Omron CX-Programmer project NewProject (CX-Programmer 9.70)

# PLC NOVO_PAP: CP1L-E EM

## Program NewProgram1 (cyclic task 0)
; POS0
Local symbols
ABRIR_LIQUIDO1 205.00 BOOL
ABRIR_LIQUIDO2 205.01 BOOL  ; ~
ABRIR_LIQUIDO3 205.02 BOOL
BIT_EXTRA1_IN 1.02 BOOL
BIT_EXTRA1_OUT 100.03 BOOL
BIT_EXTRA2_IN 1.03 BOOL
BIT_EXTRA2_OUT 100.06 BOOL
BUSY 0.06 BOOL
CONDICAO 207.01 BOOL
ENTR_1 0.07 BOOL
ENTR_2 0.08 BOOL
ENTR_3 0.09 BOOL
ENTR_4 0.10 BOOL
ENTR_5 0.11 BOOL
ENTR_6 1.00 BOOL
ENTR_7 1.01 BOOL
ENVIAR100 101.03 BOOL
ENVIAR33 101.00 BOOL
ENVIAR50 101.01 BOOL
ENVIAR66 101.02 BOOL
ENVIAR_ROBO 100.05 BOOL
ET BOOL
ET0 200.00 BOOL
ET10 200.01 BOOL  ; SVON
ET100 203.00 BOOL
ET110 203.01 BOOL
ET120 203.02 BOOL
ET130 203.03 BOOL
ET140 203.04 BOOL
ET150 203.05 BOOL
ET160 203.06 BOOL
ET170 203.07 BOOL
ET20 200.02 BOOL  ; SETUP
ET200 203.00 BOOL
ET210 203.01 BOOL
ET220 203.02 BOOL
ET230 203.03 BOOL
ET240 203.04 BOOL
ET250 203.05 BOOL
ET260 203.06 BOOL
ET30 200.03 BOOL
ET40 200.04 BOOL
ET50 200.05 BOOL
ET60 200.06 BOOL
ET70 200.07 BOOL
ET80 201.00 BOOL
ET_POS0 202.00 BOOL
ET_POS1 202.01 BOOL
ET_POS2 202.02 BOOL
ET_POS_RETORNO 202.05 BOOL
EXTRA_BIT1_IN BOOL
FAKE_IMPULSO 201.01 BOOL
IMPULSO 100.02 BOOL
IN0 100.01 BOOL
IN0W 202.03 BOOL
IN1 100.00 BOOL
IN1W 202.04 BOOL
IS_WORKING 207.02 BOOL
JA_TEM_VALOR1 203.07 BOOL
JA_TEM_VALOR2 204.04 BOOL
JA_TEM_VALOR3 204.05 BOOL
LIQUIDO1 D20 INT
LIQUIDO2 D21 INT
LIQUIDO3 D22 INT
MULT_1 D10 UINT
MULT_2 D11 UINT
MULT_3 D12 UINT
MULT_4 D13 UINT
MULT_5 D14 UINT
MULT_6 D15 UINT
MULT_7 D16 UINT
M_START 207.00 BOOL
M_STARt BOOL
NUM100 204.03 BOOL
NUM33 204.00 BOOL
NUM50 204.01 BOOL
NUM66 204.02 BOOL
OUT0 0.03 BOOL
OUT1 0.02 BOOL
POS0 201.02 BOOL
POS1 201.03 BOOL
POS1_TIMER 201.06 BOOL
POS2 201.04 BOOL
POS2_TIMER 201.07 BOOL
POS3 BOOL
POS_RASP 1.04 BOOL
POS_RASP2 1.05 BOOL
POS_RETORNO 201.05 BOOL
SETON 0.04 BOOL
SETUP 100.07 BOOL
START 0.01 BOOL
STOP 0.00 BOOL
SVON 100.04 BOOL
Start_Virtual 5.01 BOOL

### Section MAIN

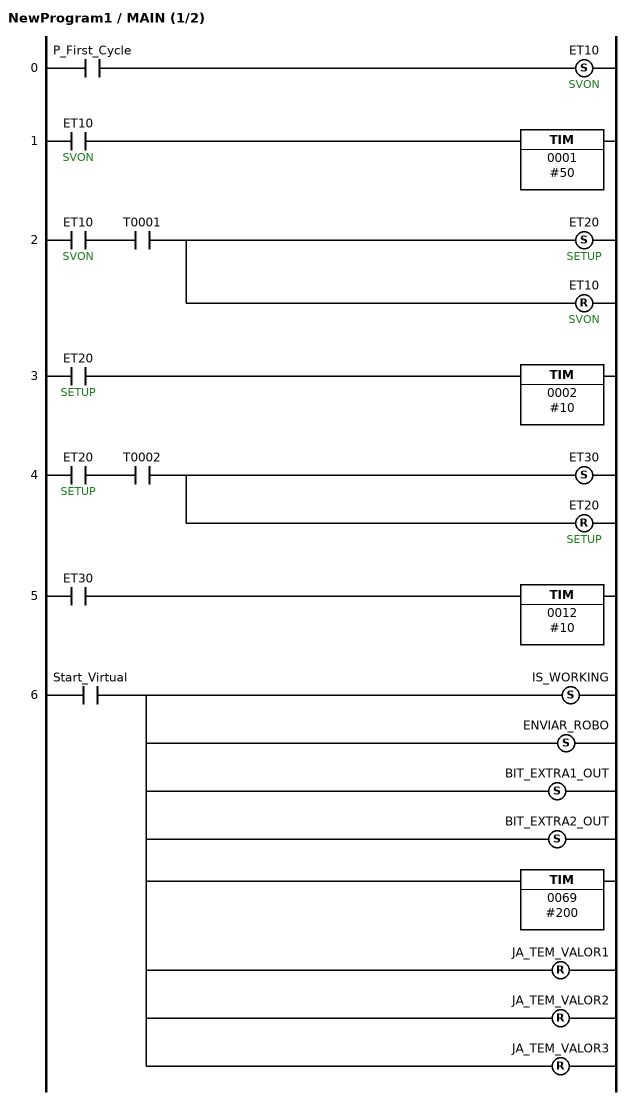
; rung 0
LD P_First_Cycle
SET ET10  ; SVON
; rung 1
LD ET10  ; SVON
TIM 0001 #50
; rung 2
LD ET10  ; SVON
AND T0001
SET ET20  ; SETUP
RSET ET10  ; SVON
; rung 3
LD ET20  ; SETUP
TIM 0002 #10
; rung 4
LD ET20  ; SETUP
AND T0002
SET ET30
RSET ET20  ; SETUP
; rung 5
LD ET30
TIM 0012 #10
; rung 6
LD Start_Virtual
SET IS_WORKING
SET ENVIAR_ROBO
SET BIT_EXTRA1_OUT
SET BIT_EXTRA2_OUT
TIM 0069 #200
RSET JA_TEM_VALOR1
RSET JA_TEM_VALOR2
RSET JA_TEM_VALOR3

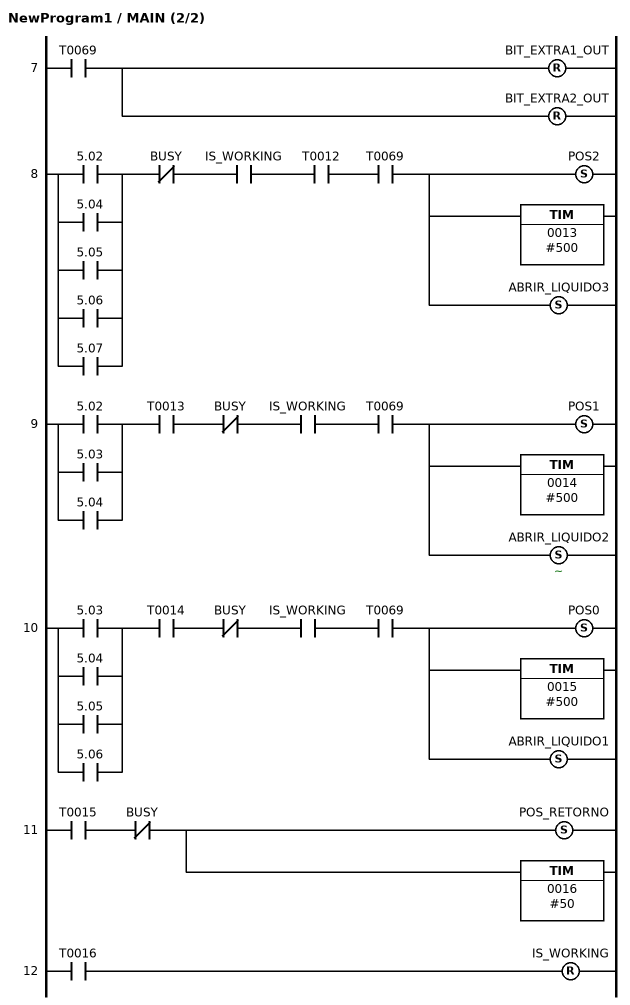
; rung 7
LD T0069
RSET BIT_EXTRA1_OUT
RSET BIT_EXTRA2_OUT
; rung 8
LD 5.02
OR 5.04
OR 5.05
OR 5.06
OR 5.07
ANDNOT BUSY
AND IS_WORKING
AND T0012
AND T0069
SET POS2
TIM 0013 #500
SET ABRIR_LIQUIDO3
; rung 9
LD 5.02
OR 5.03
OR 5.04
AND T0013
ANDNOT BUSY
AND IS_WORKING
AND T0069
SET POS1
TIM 0014 #500
SET ABRIR_LIQUIDO2  ; ~
; rung 10
LD 5.03
OR 5.04
OR 5.05
OR 5.06
AND T0014
ANDNOT BUSY
AND IS_WORKING
AND T0069
SET POS0
TIM 0015 #500
SET ABRIR_LIQUIDO1
; rung 11
LD T0015
ANDNOT BUSY
SET POS_RETORNO
TIM 0016 #50
; rung 12
LD T0016
RSET IS_WORKING

### Section SAIDAS

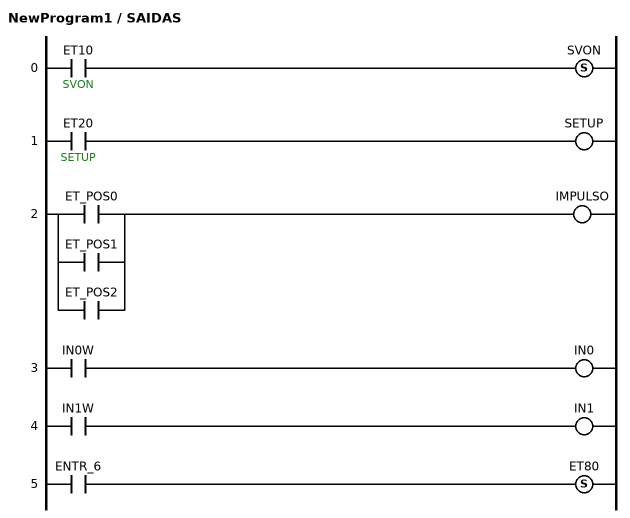
; rung 0
LD ET10  ; SVON
SET SVON
; rung 1
LD ET20  ; SETUP
OUT SETUP
; rung 2
LD ET_POS0
OR ET_POS1
OR ET_POS2
OUT IMPULSO
; rung 3
LD IN0W
OUT IN0
; rung 4
LD IN1W
OUT IN1
; rung 5
LD ENTR_6
SET ET80

### Section DE_RASP

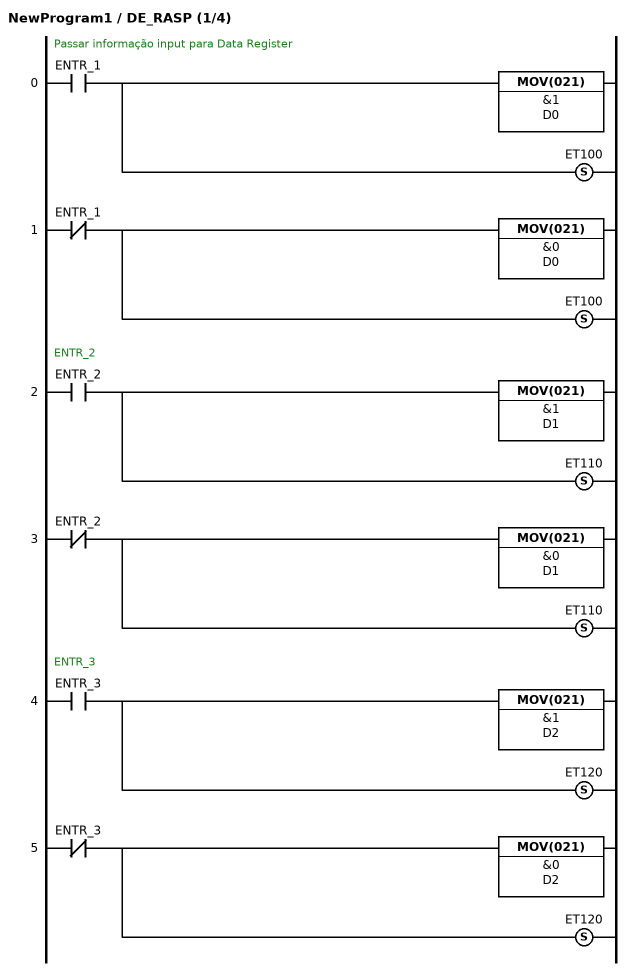
; rung 0: Passar informação input para Data Register
LD ENTR_1
MOV(021) &1 D0
SET ET100
; rung 1
LDNOT ENTR_1
MOV(021) &0 D0
SET ET100
; rung 2: ENTR_2
LD ENTR_2
MOV(021) &1 D1
SET ET110
; rung 3
LDNOT ENTR_2
MOV(021) &0 D1
SET ET110
; rung 4: ENTR_3
LD ENTR_3
MOV(021) &1 D2
SET ET120
; rung 5
LDNOT ENTR_3
MOV(021) &0 D2
SET ET120

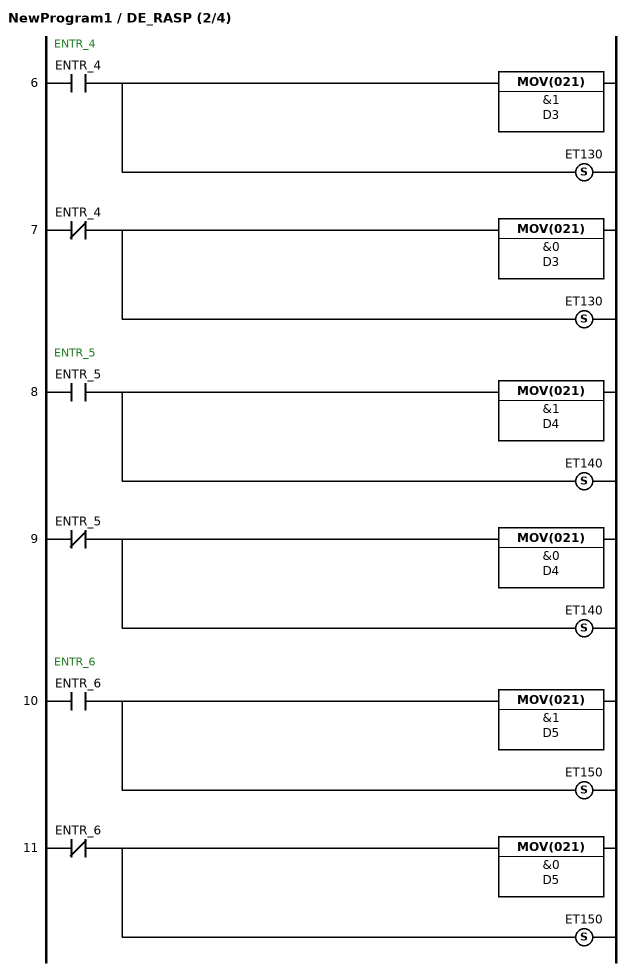
; rung 6: ENTR_4
LD ENTR_4
MOV(021) &1 D3
SET ET130
; rung 7
LDNOT ENTR_4
MOV(021) &0 D3
SET ET130
; rung 8: ENTR_5
LD ENTR_5
MOV(021) &1 D4
SET ET140
; rung 9
LDNOT ENTR_5
MOV(021) &0 D4
SET ET140
; rung 10: ENTR_6
LD ENTR_6
MOV(021) &1 D5
SET ET150
; rung 11
LDNOT ENTR_6
MOV(021) &0 D5
SET ET150

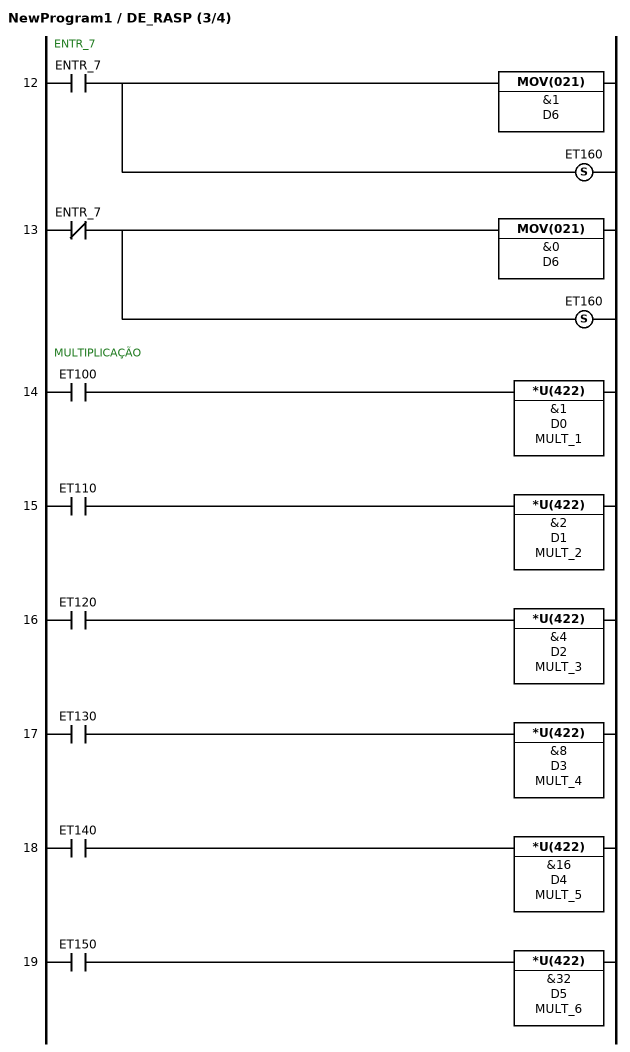
; rung 12: ENTR_7
LD ENTR_7
MOV(021) &1 D6
SET ET160
; rung 13
LDNOT ENTR_7
MOV(021) &0 D6
SET ET160
; rung 14: MULTIPLICAÇÃO
LD ET100
*U(422) &1 D0 MULT_1
; rung 15
LD ET110
*U(422) &2 D1 MULT_2
; rung 16
LD ET120
*U(422) &4 D2 MULT_3
; rung 17
LD ET130
*U(422) &8 D3 MULT_4
; rung 18
LD ET140
*U(422) &16 D4 MULT_5
; rung 19
LD ET150
*U(422) &32 D5 MULT_6

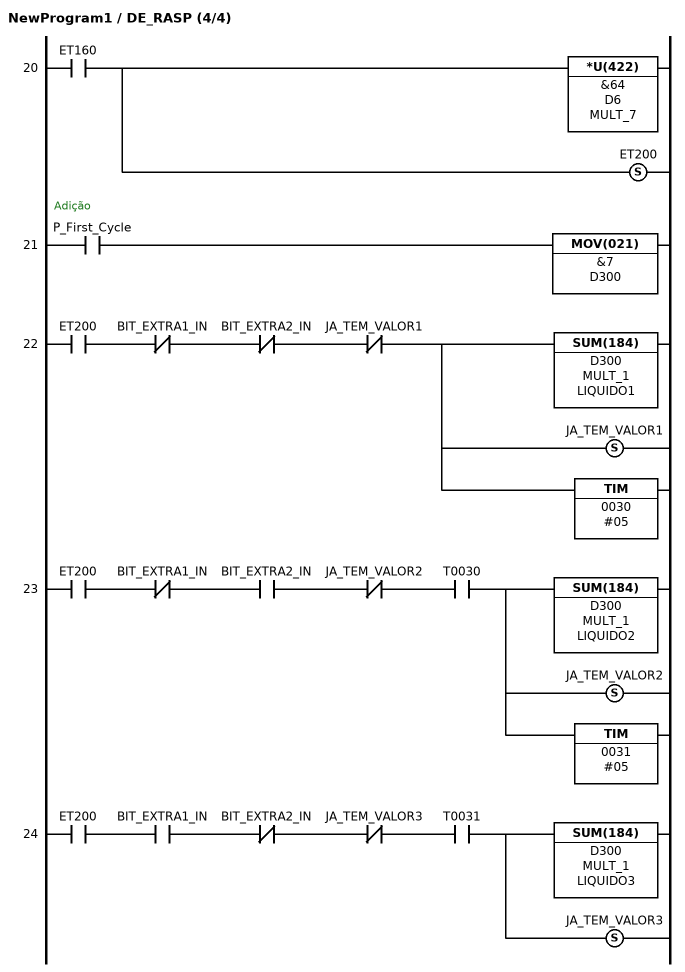
; rung 20
LD ET160
*U(422) &64 D6 MULT_7
SET ET200
; rung 21: Adição
LD P_First_Cycle
MOV(021) &7 D300
; rung 22
LD ET200
ANDNOT BIT_EXTRA1_IN
ANDNOT BIT_EXTRA2_IN
ANDNOT JA_TEM_VALOR1
SUM(184) D300 MULT_1 LIQUIDO1
SET JA_TEM_VALOR1
TIM 0030 #05
; rung 23
LD ET200
ANDNOT BIT_EXTRA1_IN
AND BIT_EXTRA2_IN
ANDNOT JA_TEM_VALOR2
AND T0030
SUM(184) D300 MULT_1 LIQUIDO2
SET JA_TEM_VALOR2
TIM 0031 #05
; rung 24
LD ET200
AND BIT_EXTRA1_IN
ANDNOT BIT_EXTRA2_IN
ANDNOT JA_TEM_VALOR3
AND T0031
SUM(184) D300 MULT_1 LIQUIDO3
SET JA_TEM_VALOR3

### Section POSIÇÕES

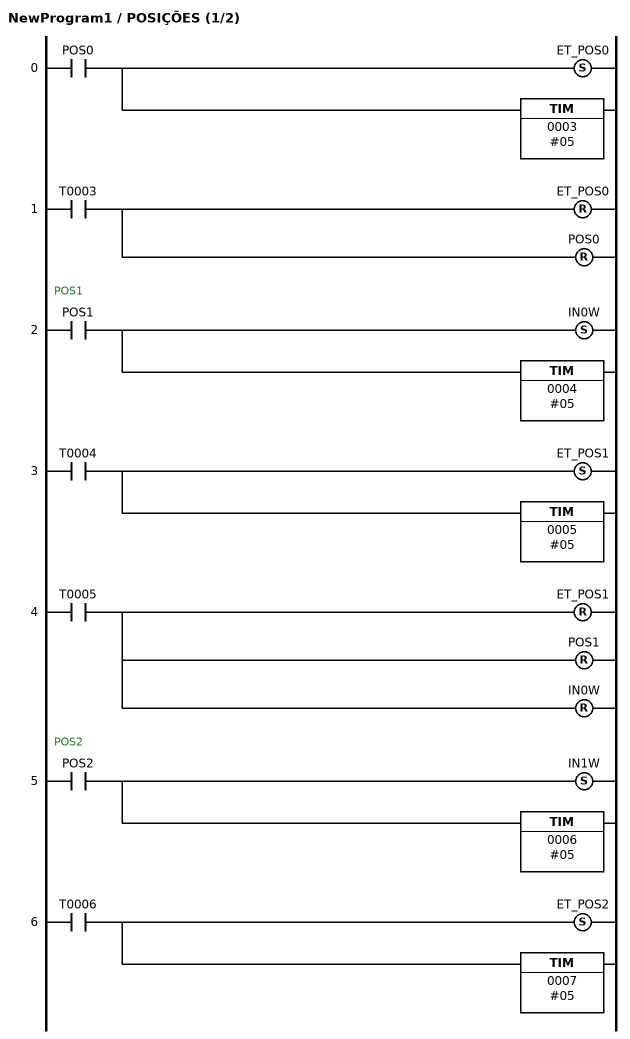
; rung 0
LD POS0
SET ET_POS0
TIM 0003 #05
; rung 1
LD T0003
RSET ET_POS0
RSET POS0
; rung 2: POS1
LD POS1
SET IN0W
TIM 0004 #05
; rung 3
LD T0004
SET ET_POS1
TIM 0005 #05
; rung 4
LD T0005
RSET ET_POS1
RSET POS1
RSET IN0W
; rung 5: POS2
LD POS2
SET IN1W
TIM 0006 #05
; rung 6
LD T0006
SET ET_POS2
TIM 0007 #05

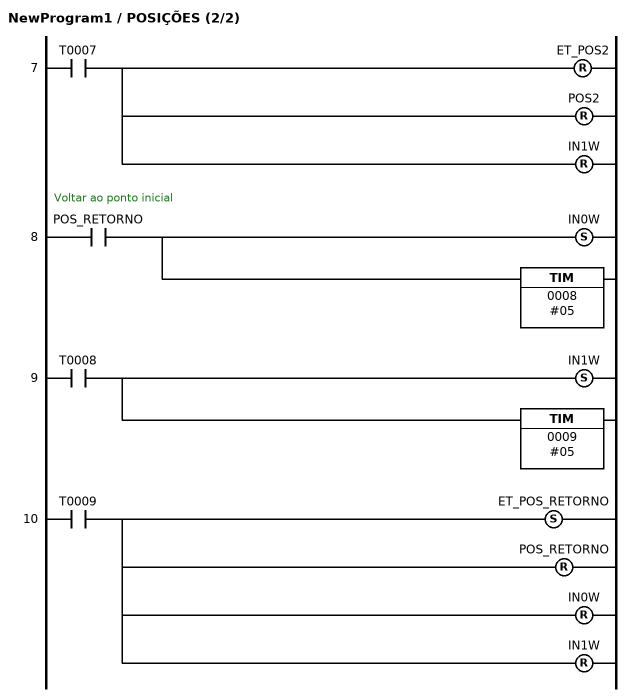
; rung 7
LD T0007
RSET ET_POS2
RSET POS2
RSET IN1W
; rung 8: Voltar ao ponto inicial
LD POS_RETORNO
SET IN0W
TIM 0008 #05
; rung 9
LD T0008
SET IN1W
TIM 0009 #05
; rung 10
LD T0009
SET ET_POS_RETORNO
RSET POS_RETORNO
RSET IN0W
RSET IN1W

### Section PARA_RASP
; 33% / 66%/ 0%

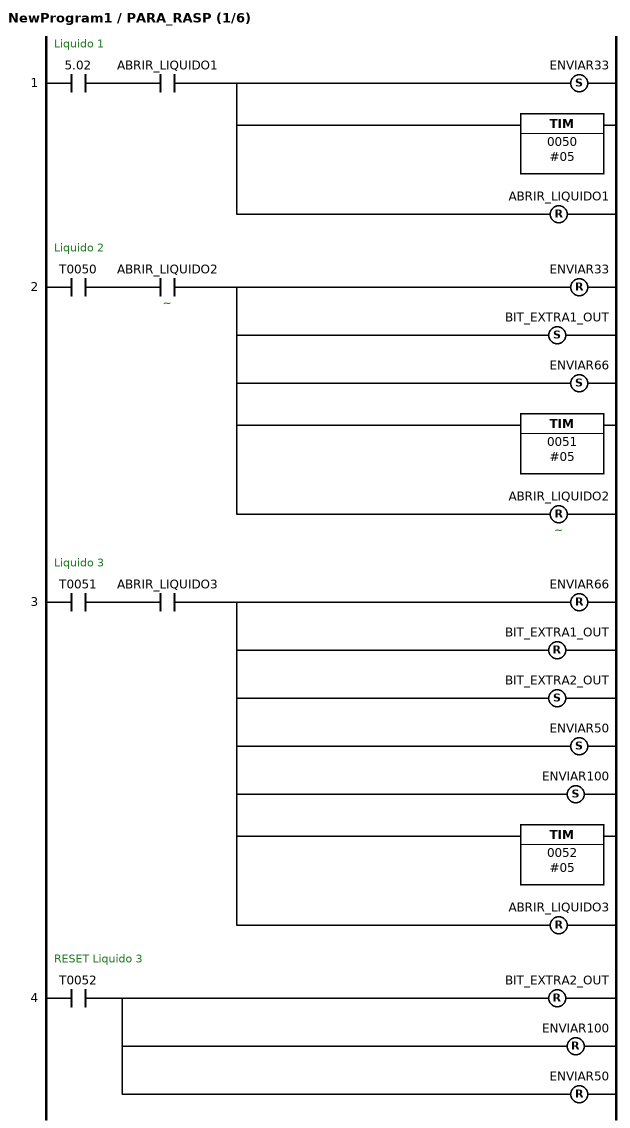
; rung 1: Liquido 1
LD 5.02
AND ABRIR_LIQUIDO1
SET ENVIAR33
TIM 0050 #05
RSET ABRIR_LIQUIDO1
; rung 2: Liquido 2
LD T0050
AND ABRIR_LIQUIDO2  ; ~
RSET ENVIAR33
SET BIT_EXTRA1_OUT
SET ENVIAR66
TIM 0051 #05
RSET ABRIR_LIQUIDO2  ; ~
; rung 3: Liquido 3
LD T0051
AND ABRIR_LIQUIDO3
RSET ENVIAR66
RSET BIT_EXTRA1_OUT
SET BIT_EXTRA2_OUT
SET ENVIAR50
SET ENVIAR100
TIM 0052 #05
RSET ABRIR_LIQUIDO3
; rung 4: RESET Liquido 3
LD T0052
RSET BIT_EXTRA2_OUT
RSET ENVIAR100
RSET ENVIAR50

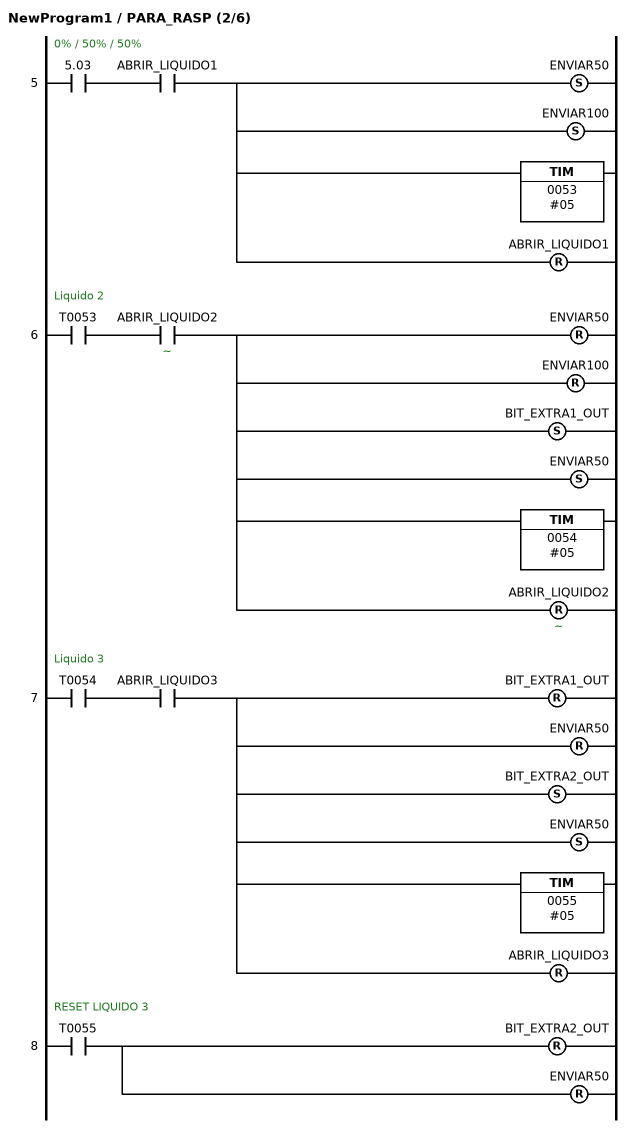
; rung 5: 0% / 50% / 50%
LD 5.03
AND ABRIR_LIQUIDO1
SET ENVIAR50
SET ENVIAR100
TIM 0053 #05
RSET ABRIR_LIQUIDO1
; rung 6: Liquido 2
LD T0053
AND ABRIR_LIQUIDO2  ; ~
RSET ENVIAR50
RSET ENVIAR100
SET BIT_EXTRA1_OUT
SET ENVIAR50
TIM 0054 #05
RSET ABRIR_LIQUIDO2  ; ~
; rung 7: Liquido 3
LD T0054
AND ABRIR_LIQUIDO3
RSET BIT_EXTRA1_OUT
RSET ENVIAR50
SET BIT_EXTRA2_OUT
SET ENVIAR50
TIM 0055 #05
RSET ABRIR_LIQUIDO3
; rung 8: RESET LIQUIDO 3
LD T0055
RSET BIT_EXTRA2_OUT
RSET ENVIAR50

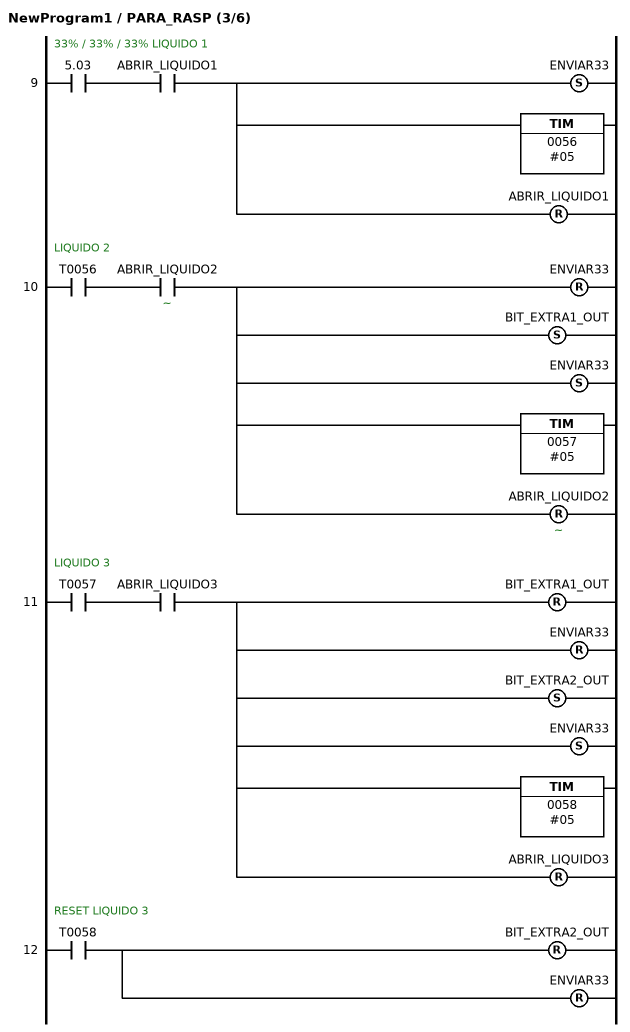
; rung 9: 33% / 33% / 33% LIQUIDO 1
LD 5.03
AND ABRIR_LIQUIDO1
SET ENVIAR33
TIM 0056 #05
RSET ABRIR_LIQUIDO1
; rung 10: LIQUIDO 2
LD T0056
AND ABRIR_LIQUIDO2  ; ~
RSET ENVIAR33
SET BIT_EXTRA1_OUT
SET ENVIAR33
TIM 0057 #05
RSET ABRIR_LIQUIDO2  ; ~
; rung 11: LIQUIDO 3
LD T0057
AND ABRIR_LIQUIDO3
RSET BIT_EXTRA1_OUT
RSET ENVIAR33
SET BIT_EXTRA2_OUT
SET ENVIAR33
TIM 0058 #05
RSET ABRIR_LIQUIDO3
; rung 12: RESET LIQUIDO 3
LD T0058
RSET BIT_EXTRA2_OUT
RSET ENVIAR33

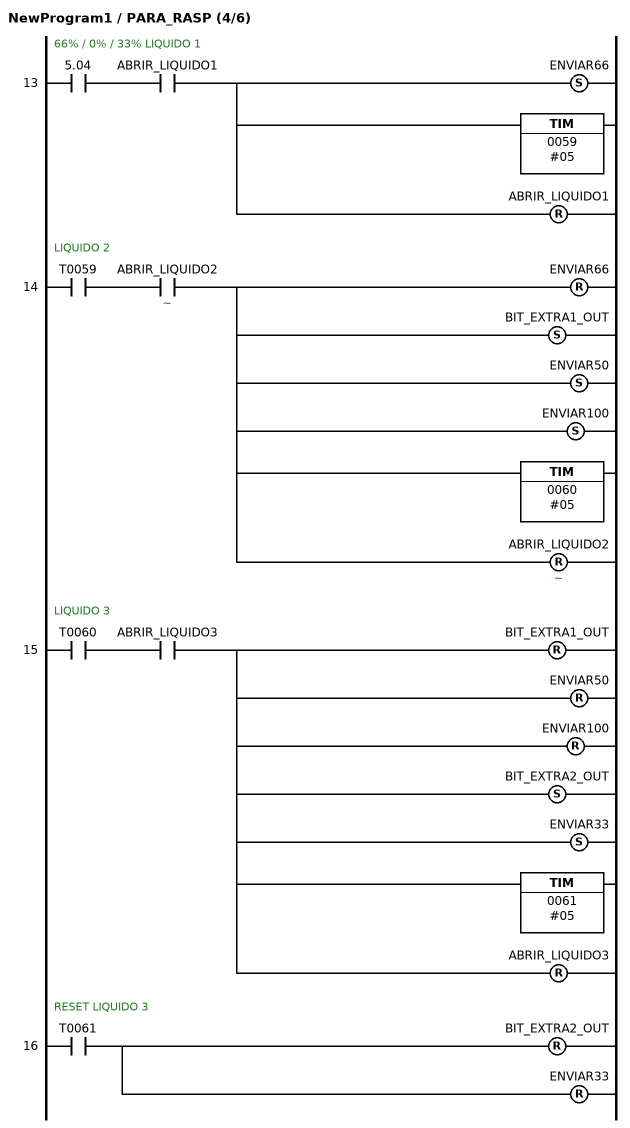
; rung 13: 66% / 0% / 33% LIQUIDO 1
LD 5.04
AND ABRIR_LIQUIDO1
SET ENVIAR66
TIM 0059 #05
RSET ABRIR_LIQUIDO1
; rung 14: LIQUIDO 2
LD T0059
AND ABRIR_LIQUIDO2  ; ~
RSET ENVIAR66
SET BIT_EXTRA1_OUT
SET ENVIAR50
SET ENVIAR100
TIM 0060 #05
RSET ABRIR_LIQUIDO2  ; ~
; rung 15: LIQUIDO 3
LD T0060
AND ABRIR_LIQUIDO3
RSET BIT_EXTRA1_OUT
RSET ENVIAR50
RSET ENVIAR100
SET BIT_EXTRA2_OUT
SET ENVIAR33
TIM 0061 #05
RSET ABRIR_LIQUIDO3
; rung 16: RESET LIQUIDO 3
LD T0061
RSET BIT_EXTRA2_OUT
RSET ENVIAR33

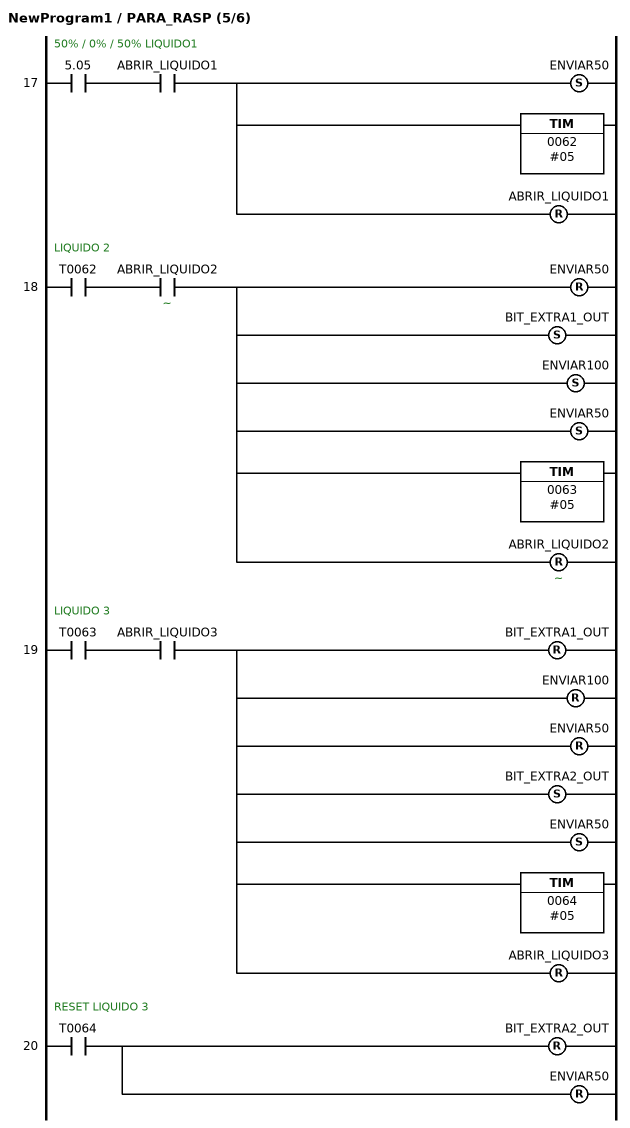
; rung 17: 50% / 0% / 50% LIQUIDO1
LD 5.05
AND ABRIR_LIQUIDO1
SET ENVIAR50
TIM 0062 #05
RSET ABRIR_LIQUIDO1
; rung 18: LIQUIDO 2
LD T0062
AND ABRIR_LIQUIDO2  ; ~
RSET ENVIAR50
SET BIT_EXTRA1_OUT
SET ENVIAR100
SET ENVIAR50
TIM 0063 #05
RSET ABRIR_LIQUIDO2  ; ~
; rung 19: LIQUIDO 3
LD T0063
AND ABRIR_LIQUIDO3
RSET BIT_EXTRA1_OUT
RSET ENVIAR100
RSET ENVIAR50
SET BIT_EXTRA2_OUT
SET ENVIAR50
TIM 0064 #05
RSET ABRIR_LIQUIDO3
; rung 20: RESET LIQUIDO 3
LD T0064
RSET BIT_EXTRA2_OUT
RSET ENVIAR50

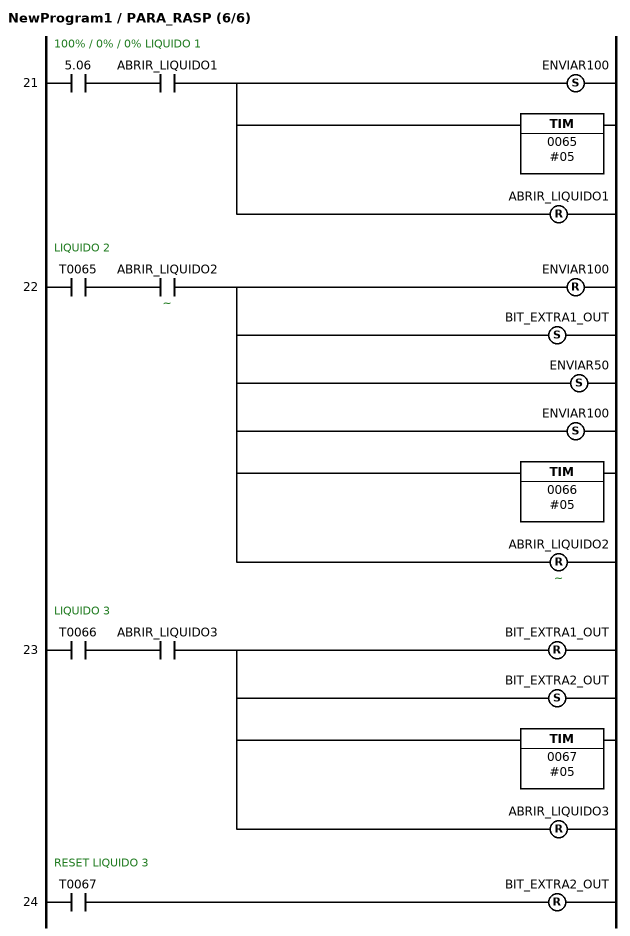
; rung 21: 100% / 0% / 0% LIQUIDO 1
LD 5.06
AND ABRIR_LIQUIDO1
SET ENVIAR100
TIM 0065 #05
RSET ABRIR_LIQUIDO1
; rung 22: LIQUIDO 2
LD T0065
AND ABRIR_LIQUIDO2  ; ~
RSET ENVIAR100
SET BIT_EXTRA1_OUT
SET ENVIAR50
SET ENVIAR100
TIM 0066 #05
RSET ABRIR_LIQUIDO2  ; ~
; rung 23: LIQUIDO 3
LD T0066
AND ABRIR_LIQUIDO3
RSET BIT_EXTRA1_OUT
SET BIT_EXTRA2_OUT
TIM 0067 #05
RSET ABRIR_LIQUIDO3
; rung 24: RESET LIQUIDO 3
LD T0067
RSET BIT_EXTRA2_OUT

### Section RASP_EIXO

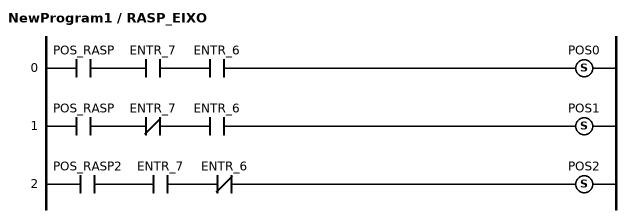
; rung 0
LD POS_RASP
AND ENTR_7
AND ENTR_6
SET POS0
; rung 1
LD POS_RASP
ANDNOT ENTR_7
AND ENTR_6
SET POS1
; rung 2
LD POS_RASP2
AND ENTR_7
ANDNOT ENTR_6
SET POS2

### Section END
; rung 0
END(001)